TYPE ST_GantryProdPar :
STRUCT
	PositionHorizontalPickup			: LREAL;
	PositionHorizontalDropOff			: LREAL;
	PositionVerticalPickup				: LREAL;
	PositionVerticalDropOff				: LREAL;
	
	BlowOffTime							: TIME;
	
END_STRUCT
END_TYPE

(* stored: Version 1.1.0.1, ProductVersion 3.1.4020.12
   DUT ST_GantryProdPar: Id {9869e799-f671-4a1f-a0ab-0f8d1e6b503b} *)
